FUNCTION "FC_Off_Dly_T_0.1s" : VOID
TITLE =%version: 0.03 % CN: 30
//Function:
//This function create an off delay on the signal "Start".
//
//Description:
//The output signal "Status" will be high on the input signal "Start" and if
//the off delay is not elapsed.
//The count of the delay time is only done while "Enable" is high. So you can use
//this as a retentive timer.
//
//Off-delay time characteristics:
//
//                             |<-- t -->|
//                    _________
//Start input    ____|         |______________
//
//                              _________
//Timer running  ______________|         |____
//
//                    ___________________
//Status         ____|                   |____
//
//
//
//DECREMENT:
//The counter is decremented by one if the signal state at input
//Start="0" and Enable="1" on every 0.1sec one-shot and the value of
//the counter is greater than "0".
//
//SET:
//The Counter is preset with the value at input Time_Value if input Start="1".
//Time_Value only accept if >=0 and <=32767 else the counter is preset with 0.
//If Set Off-delay and the Time_Value is not accepted the BR will be "0".
//This indicate an error occurred during execution, the BR bit is "0".
//If the function was executed with no error, the BR bit is "1".
//
//Time_Value format [* 0.1 Sec]
//
//STATUS:
//The signal state at output status is "1" if
//start="1' and if Start='0' the counter is not equal to zero. This mains the
//off delay time not is elapesed.
//
//History:
//This version  %created_by: nlhdl %
//              %date_created: maandag 6 juli 2015 10:28:31 %
//              %release: VI_CONV/RA_Dev_Oakham %
//
//Modification History:                                   By:    Date:     Rev:
//----------------------------------------------------  -------  --------  -----
//7324: ECS-P General from the RD to RA for platform    nlHdL    06-07-15   0.03
//14163: Removed IO parameter added In- or Output       nlHdL    06-01-14   0.03
//15807: Block consistency update IO symbols, comment   nlHdL    18-09-13   0.02
//Copied from SSS                                         nlHdL  11-01-11   0.01
//Based on FC_Off_Dly_T_0.1s 1.5
//
//
FAMILY : General
VERSION : 0.0


VAR_INPUT
  i_Start : BOOL ;	//Start count
  i_Enable_Dly : BOOL ;	//Enable delay timer
  i_Time_Value : INT ;	//[0.1 sec] Preset Value
  i_Current_Value : INT ;	//[0.1 sec] Current counter value
END_VAR
VAR_OUTPUT
  o_Status : BOOL ;	//Delay counter active count >0
  o_Current_Value : INT ;	//Current counter value
END_VAR
VAR_TEMP
  t_Elapsed : BOOL ;	//Timer elapsed
  t_Current_Value : INT ;	//Temp Current counter value
END_VAR
BEGIN
NETWORK
TITLE =AA: Init BR Binary Result Bit
// Init the BR-bit as a good result
      SET   ; // Init
      SAVE  ; // BR-bit
NETWORK
TITLE =BA: Counter down
//If 'Start' and Enable and time_one_shot the counter will decrement.
//In the network 'Counter status' the counter will be kept to zero if
//the counter become < "0". So the counter will not be negative.
      L     #i_Current_Value;
      T     #t_Current_Value;

      AN    #i_Start; // IF   count down
      A     #i_Enable_Dly; // AND  enable
      A     "M_OS_/0.1_sec."; // AND  time_one_shot
      JCN   BA99; // ELSE no count
      L     #t_Current_Value; // THEN currunt value-1
      +     -1;
      T     #t_Current_Value;
BA99: NOP   0;
NETWORK
TITLE =CA: Preset counter
//IF 'START' then preset counter
//IF 'Preset_Value' is between 0 and 32767 (max integer)
//the counter take over the preset value into 'Current_Value'
//else the 'Current-Value' will be zero.
//IF preset and the "Time_Value" is out of range then the BR-bit will be "0".
      A     #i_Start; // IF   set counter
      JCN   CA99; // ELSE no preset
      L     32767; // Max preset value
      L     #i_Time_Value; // Preset value
      >=I   ; // IF   lower or same max
      A(    ; // AND
      L     0; // Min preset value
      >=I   ; // IF   higher or same min
      )     ;
      SAVE  ; // IF Accept Time_Value THEN BR="1" ELSE BR="0"
      JCN   CA01; // ELSE preset zero
      L     #i_Time_Value; // THEN time_value
CA01: T     #t_Current_Value; // Preset: Current value
CA99: NOP   0;
NETWORK
TITLE =DA: Counter status
//If the counter <= "0" the time has elapsed
//The counter can not be negative so it will be kept to zero
      L     #t_Current_Value; // IF   current value counter = 0
      L     0;
      <=I   ;
      =     #t_Elapsed; // THEN time elapesed so status := '1'
      JCN   DA99;
      T     #t_Current_Value; // ALSO keep counter zero
DA99: NOP   0;
NETWORK
TITLE =EA: (..) Off-delay status
//Status off-delay
      L     #t_Current_Value;
      T     #o_Current_Value;

      O     #i_Start; // IF   'Start'
      ON    #t_Elapsed; // OR   off_delay time is not elepsed
      =     #o_Status; // THEN status := '1'
END_FUNCTION

